(* IEC 61131-3 sources: cybercode_codesys_lib/src/signal/Analog, 5 files *)

(* ---- E_AlarmSetpoints.st ---- *)
TYPE E_AlarmSetpoints :
(
	Normal 	:= 0,
	L		:= 1,
	H		:= 2,
	LL		:= 3,
	HH		:= 4
);
END_TYPE

(* ---- FB_AnalogSignal4_20mA.st ---- *)
FUNCTION_BLOCK FB_AnalogSignal4_20mA EXTENDS FB_BasicAnalogSignal
VAR_INPUT
    rScaleMin : REAL := 0.0;        // Минимальное значение масштабируемого диапазона
    rScaleMax : REAL := 100.0;      // Максимальное значение масштабируемого диапазона
    xEnableRangeProtection : BOOL := TRUE;  // Включение защиты от выхода за диапазон
END_VAR
VAR_OUTPUT
END_VAR
VAR
    // Константы для токовой петли 4..20 мА
    _rCurrentMin : REAL := 4.0;     // Минимальный ток (мА)
    _rCurrentMax : REAL := 20.0;    // Максимальный ток (мА)

    // Состояние сигнала
    _xUnderrange : BOOL := FALSE;   // Сигнал ниже 4 мА
    _xOverrange : BOOL := FALSE;    // Сигнал выше 20 мА
    _xWireBreak : BOOL := FALSE;    // Обрыв линии (ток < 3.5 мА)
    _xOverload : BOOL := FALSE;     // Перегрузка (ток > 21 мА)

    // Пороговые значения для диагностики
    _rWireBreakThreshold : REAL := 3.5;    // Порог обрыва линии
    _rOverloadThreshold : REAL := 21.0;    // Порог перегрузки
END_VAR

// =====================================
// INPUT PROCESSING
// =====================================
ProcessRawValue();

// =====================================
// MAIN LOGIC
// =====================================
DiagnoseCurrent();

(* Обработка исходного токового сигнала *)
METHOD ProcessRawValue
VAR_INPUT
END_VAR
VAR
    rNormalizedCurrent : REAL;
END_VAR
    // Нормализация тока в диапазон 0..1
    IF (_rCurrentMax - _rCurrentMin) <> 0 THEN
        rNormalizedCurrent := (GetRawValue() - _rCurrentMin) / (_rCurrentMax - _rCurrentMin);
    ELSE
        rNormalizedCurrent := 0.0;
    END_IF

    // Масштабирование к заданному диапазону
    IF xEnableRangeProtection THEN
        // С ограничением диапазона
        rNormalizedCurrent := ClampToRange01(rNormalizedCurrent);
    END_IF

    SetProcessedValue(rScaleMin + rNormalizedCurrent * (rScaleMax - rScaleMin));
END_METHOD

(* Диагностика токового сигнала *)
METHOD PRIVATE DiagnoseCurrent
VAR_INPUT
END_VAR
VAR
    rCurrentValue : REAL;
END_VAR
    rCurrentValue := GetRawValue();

    // Проверка на обрыв линии
    _xWireBreak := rCurrentValue < _rWireBreakThreshold;

    // Проверка на перегрузку
    _xOverload := rCurrentValue > _rOverloadThreshold;

    // Проверка на выход за рабочий диапазон 4..20 мА
    _xUnderrange := (rCurrentValue < _rCurrentMin) AND NOT _xWireBreak;
    _xOverrange := (rCurrentValue > _rCurrentMax) AND NOT _xOverload;
END_METHOD

(* Получение масштабированного значения с учетом ошибок *)
METHOD GetScaledValue : REAL
VAR_INPUT
END_VAR
    IF _xWireBreak OR _xOverload THEN
        // При критических ошибках возвращаем минимальное значение
        GetScaledValue := rScaleMin;
    ELSE
        GetScaledValue := GetProcessedValue();
    END_IF
END_METHOD

(* Получение процентного значения (0..100%) *)
METHOD GetPercentValue : REAL
VAR_INPUT
END_VAR
VAR
    rNormalized : REAL;
END_VAR
    IF (rScaleMax - rScaleMin) <> 0 THEN
        rNormalized := (GetProcessedValue() - rScaleMin) / (rScaleMax - rScaleMin);
        GetPercentValue := rNormalized * 100.0;
    ELSE
        GetPercentValue := 0.0;
    END_IF
END_METHOD

(* Проверка на обрыв линии *)
METHOD IsWireBreak : BOOL
VAR_INPUT
END_VAR
    IsWireBreak := _xWireBreak;
END_METHOD

(* Проверка на перегрузку *)
METHOD IsOverload : BOOL
VAR_INPUT
END_VAR
    IsOverload := _xOverload;
END_METHOD

(* Проверка на нижний предел диапазона *)
METHOD IsUnderrange : BOOL
VAR_INPUT
END_VAR
    IsUnderrange := _xUnderrange;
END_METHOD

(* Проверка на верхний предел диапазона *)
METHOD IsOverrange : BOOL
VAR_INPUT
END_VAR
    IsOverrange := _xOverrange;
END_METHOD

(* Проверка на любую ошибку *)
METHOD HasError : BOOL
VAR_INPUT
END_VAR
    HasError := _xWireBreak OR _xOverload OR _xUnderrange OR _xOverrange;
END_METHOD

(* Установка масштабируемого диапазона *)
METHOD SetScaleRange
VAR_INPUT
    rMin : REAL;
    rMax : REAL;
END_VAR
    IF rMin < rMax THEN
        rScaleMin := rMin;
        rScaleMax := rMax;
    END_IF
END_METHOD

(* Получение минимального масштабируемого значения *)
METHOD GetScaleMin : REAL
VAR_INPUT
END_VAR
    GetScaleMin := rScaleMin;
END_METHOD

(* Получение максимального масштабируемого значения *)
METHOD GetScaleMax : REAL
VAR_INPUT
END_VAR
    GetScaleMax := rScaleMax;
END_METHOD

(* Сброс всех ошибок и состояний *)
METHOD Reset
VAR_INPUT
END_VAR
    // Вызов родительского сброса
    SUPER^.Reset();

    // Сброс локальных флагов
    _xUnderrange := FALSE;
    _xOverrange := FALSE;
    _xWireBreak := FALSE;
    _xOverload := FALSE;
END_METHOD

(* ========================================
   ЗАЩИЩЕННЫЕ МЕТОДЫ
   ======================================== *)

(* Ограничение значения в диапазоне 0..1 *)
METHOD PROTECTED ClampToRange01 : REAL
VAR_INPUT
    rValue : REAL;
END_VAR
    IF rValue < 0.0 THEN
        ClampToRange01 := 0.0;
    ELSIF rValue > 1.0 THEN
        ClampToRange01 := 1.0;
    ELSE
        ClampToRange01 := rValue;
    END_IF
END_METHOD

END_FUNCTION_BLOCK

(* ---- FB_BasicAnalogSignal.st ---- *)
FUNCTION_BLOCK ABSTRACT FB_BasicAnalogSignal
VAR_INPUT
    irRawValue : REAL;          // Исходное значение аналогового сигнала
END_VAR
VAR_OUTPUT
END_VAR
VAR
    _rProcessedValue : REAL;    // Обработанное значение сигнала
    _rMinValue : REAL := 0.0;   // Минимальное допустимое значение
    _rMaxValue : REAL := 100.0; // Максимальное допустимое значение
    _xOutOfRange : BOOL := FALSE; // Флаг выхода за пределы диапазона
END_VAR

// =====================================
// INPUT PROCESSING
// =====================================
ProcessRawValue();

// =====================================
// MAIN LOGIC
// =====================================
ValidateRange();

(* Получение исходного значения *)
METHOD GetRawValue : REAL
VAR_INPUT
END_VAR
    GetRawValue := irRawValue;
END_METHOD

(* Получение обработанного значения *)
METHOD GetProcessedValue : REAL
VAR_INPUT
END_VAR
    GetProcessedValue := _rProcessedValue;
END_METHOD

(* Получение статуса выхода за пределы диапазона *)
METHOD IsOutOfRange : BOOL
VAR_INPUT
END_VAR
    IsOutOfRange := _xOutOfRange;
END_METHOD

(* Получение минимального значения диапазона *)
METHOD GetMinValue : REAL
VAR_INPUT
END_VAR
    GetMinValue := _rMinValue;
END_METHOD

(* Получение максимального значения диапазона *)
METHOD GetMaxValue : REAL
VAR_INPUT
END_VAR
    GetMaxValue := _rMaxValue;
END_METHOD

(* Установка диапазона допустимых значений *)
METHOD SetRange
VAR_INPUT
    rMinValue : REAL;
    rMaxValue : REAL;
END_VAR
    IF rMinValue < rMaxValue THEN
        _rMinValue := rMinValue;
        _rMaxValue := rMaxValue;
    END_IF
END_METHOD

(* Проверка принадлежности значения к диапазону *)
METHOD IsInRange : BOOL
VAR_INPUT
    rValue : REAL;
END_VAR
    IsInRange := (rValue >= _rMinValue) AND (rValue <= _rMaxValue);
END_METHOD

(* Ограничение значения в пределах диапазона *)
METHOD ClampToRange : REAL
VAR_INPUT
    rValue : REAL;
END_VAR
    IF rValue < _rMinValue THEN
        ClampToRange := _rMinValue;
    ELSIF rValue > _rMaxValue THEN
        ClampToRange := _rMaxValue;
    ELSE
        ClampToRange := rValue;
    END_IF
END_METHOD

(* Сброс состояния функционального блока *)
METHOD Reset
VAR_INPUT
END_VAR
    _rProcessedValue := 0.0;
    _xOutOfRange := FALSE;
END_METHOD

(* ========================================
   АБСТРАКТНЫЕ МЕТОДЫ (должны быть переопределены в наследниках)
   ======================================== *)

(* Обработка исходного значения (абстрактный метод) *)
METHOD ABSTRACT ProcessRawValue
VAR_INPUT
END_VAR
END_METHOD

(* ========================================
   ЗАЩИЩЕННЫЕ МЕТОДЫ (для использования в наследниках)
   ======================================== *)

(* Проверка диапазона значений *)
METHOD PROTECTED ValidateRange
VAR_INPUT
END_VAR
    _xOutOfRange := NOT IsInRange(_rProcessedValue);
END_METHOD

(* Установка обработанного значения *)
METHOD PROTECTED SetProcessedValue
VAR_INPUT
    rValue : REAL;
END_VAR
    _rProcessedValue := rValue;
END_METHOD

END_FUNCTION_BLOCK

(* ---- FB_RangeDiagnostic_LH.st ---- *)
FUNCTION_BLOCK FB_RangeDiagnostic_LH
VAR_INPUT
    irValue : REAL;                     // Входное значение для контроля
    irSetpointL : REAL;         		// Уставка предупреждения низкого уровня
    irSetpointLL : REAL;        		// Уставка аварии низкого уровня
    irSetpointH : REAL;         		// Уставка предупреждения высокого уровня
    irSetpointHH : REAL;        		// Уставка аварии высокого уровня
    ixEnable : BOOL := TRUE;            // Разрешение работы блока
    irHysteresis : REAL := 1.0;         // Гистерезис для предотвращения дребезга
END_VAR
VAR_OUTPUT
    quAlarmCode : E_AlarmSetpoints;     // Код текущего состояния аварии/предупреждения
    qxAlarmActive : BOOL;               // TRUE = активна любая авария или предупреждение
    qxWarningActive : BOOL;             // TRUE = активно предупреждение (L или H)
    qxCriticalActive : BOOL;            // TRUE = активна критическая авария (LL или HH)
END_VAR
VAR
    _uPreviousAlarmCode : E_AlarmSetpoints := E_AlarmSetpoints.Normal;  // Предыдущий код аварии
    _xValidSetpoints : BOOL := TRUE;                                    // Флаг корректности уставок
    _rHysteresisValue : REAL;                                          // Текущее значение гистерезиса
END_VAR

// =====================================
// ВАЛИДАЦИЯ УСТАВОК
// =====================================
ValidateSetpoints();

// =====================================
// ОСНОВНАЯ ЛОГИКА ОПРЕДЕЛЕНИЯ АВАРИЙ
// =====================================
IF ixEnable AND _xValidSetpoints THEN
    ProcessAlarms();
ELSE
    // При отключении или некорректных уставках - сброс в нормальное состояние
    quAlarmCode := E_AlarmSetpoints.Normal;
END_IF

// =====================================
// ОБНОВЛЕНИЕ ВЫХОДНЫХ СИГНАЛОВ
// =====================================
UpdateOutputs();

(* Валидация корректности уставок *)
METHOD PRIVATE ValidateSetpoints
VAR_INPUT
END_VAR
    // Проверяем логическую корректность уставок: LL < L < H < HH
    _xValidSetpoints := (irSetpointLL <= irSetpointL) AND
                       (irSetpointL < irSetpointH) AND
                       (irSetpointH <= irSetpointHH);

    // Гистерезис не может быть отрицательным
    IF irHysteresis < 0 THEN
        _rHysteresisValue := 0;
    ELSE
        _rHysteresisValue := irHysteresis;
    END_IF
END_METHOD

(* Основная логика обработки аварий с гистерезисом *)
METHOD PRIVATE ProcessAlarms
VAR_INPUT
END_VAR
    // Сохраняем предыдущее состояние
    _uPreviousAlarmCode := quAlarmCode;

    // Определяем новое состояние на основе текущего значения
    IF irValue <= irSetpointLL THEN
        quAlarmCode := E_AlarmSetpoints.LL;
    ELSIF irValue <= irSetpointL THEN
        quAlarmCode := E_AlarmSetpoints.L;
    ELSIF irValue >= irSetpointHH THEN
        quAlarmCode := E_AlarmSetpoints.HH;
    ELSIF irValue >= irSetpointH THEN
        quAlarmCode := E_AlarmSetpoints.H;
    ELSE
        // Проверяем гистерезис для возврата в нормальное состояние
        ApplyHysteresis();
    END_IF
END_METHOD

(* Применение гистерезиса для предотвращения дребезга *)
METHOD PRIVATE ApplyHysteresis
VAR_INPUT
END_VAR
    // Применяем гистерезис только при возврате к нормальному состоянию
    CASE _uPreviousAlarmCode OF
        E_AlarmSetpoints.LL:
            // Возврат из LL возможен только при превышении LL + гистерезис
            IF irValue > (irSetpointLL + _rHysteresisValue) THEN
                quAlarmCode := E_AlarmSetpoints.Normal;
            ELSE
                quAlarmCode := E_AlarmSetpoints.LL;
            END_IF

        E_AlarmSetpoints.L:
            // Возврат из L возможен только при превышении L + гистерезис
            IF irValue > (irSetpointL + _rHysteresisValue) THEN
                quAlarmCode := E_AlarmSetpoints.Normal;
            ELSE
                quAlarmCode := E_AlarmSetpoints.L;
            END_IF

        E_AlarmSetpoints.H:
            // Возврат из H возможен только при снижении ниже H - гистерезис
            IF irValue < (irSetpointH - _rHysteresisValue) THEN
                quAlarmCode := E_AlarmSetpoints.Normal;
            ELSE
                quAlarmCode := E_AlarmSetpoints.H;
            END_IF

        E_AlarmSetpoints.HH:
            // Возврат из HH возможен только при снижении ниже HH - гистерезис
            IF irValue < (irSetpointHH - _rHysteresisValue) THEN
                quAlarmCode := E_AlarmSetpoints.Normal;
            ELSE
                quAlarmCode := E_AlarmSetpoints.HH;
            END_IF

        E_AlarmSetpoints.Normal:
            // Остаемся в нормальном состоянии
            quAlarmCode := E_AlarmSetpoints.Normal;
    END_CASE
END_METHOD

(* Обновление выходных сигналов *)
METHOD PRIVATE UpdateOutputs
VAR_INPUT
END_VAR
    // Флаг активности любой аварии или предупреждения
    qxAlarmActive := (quAlarmCode <> E_AlarmSetpoints.Normal);

    // Флаг активности предупреждений (L, H)
    qxWarningActive := (quAlarmCode = E_AlarmSetpoints.L) OR
                      (quAlarmCode = E_AlarmSetpoints.H);

    // Флаг активности критических аварий (LL, HH)
    qxCriticalActive := (quAlarmCode = E_AlarmSetpoints.LL) OR
                       (quAlarmCode = E_AlarmSetpoints.HH);
END_METHOD

(* ========================================
   МЕТОДЫ ПОЛУЧЕНИЯ ИНФОРМАЦИИ
   ======================================== *)

(* Получение текущего кода аварии *)
METHOD GetAlarmCode : E_AlarmSetpoints
VAR_INPUT
END_VAR
    GetAlarmCode := quAlarmCode;
END_METHOD

(* Получение входного значения *)
METHOD GetCurrentValue : REAL
VAR_INPUT
END_VAR
    GetCurrentValue := irValue;
END_METHOD

(* Проверка состояния "в норме" *)
METHOD IsNormal : BOOL
VAR_INPUT
END_VAR
    IsNormal := (quAlarmCode = E_AlarmSetpoints.Normal);
END_METHOD

(* Проверка активности низких аварий (L или LL) *)
METHOD IsLowAlarm : BOOL
VAR_INPUT
END_VAR
    IsLowAlarm := (quAlarmCode = E_AlarmSetpoints.L) OR
                  (quAlarmCode = E_AlarmSetpoints.LL);
END_METHOD

(* Проверка активности высоких аварий (H или HH) *)
METHOD IsHighAlarm : BOOL
VAR_INPUT
END_VAR
    IsHighAlarm := (quAlarmCode = E_AlarmSetpoints.H) OR
                   (quAlarmCode = E_AlarmSetpoints.HH);
END_METHOD

(* Проверка корректности уставок *)
METHOD AreSetpointsValid : BOOL
VAR_INPUT
END_VAR
    AreSetpointsValid := _xValidSetpoints;
END_METHOD

(* Получение расстояния до ближайшей уставки *)
METHOD GetDistanceToNearestSetpoint : REAL
VAR_INPUT
END_VAR
VAR
    rDistanceToL : REAL;
    rDistanceToLL : REAL;
    rDistanceToH : REAL;
    rDistanceToHH : REAL;
    rMinDistance : REAL;
END_VAR
    rDistanceToL := ABS(irValue - irSetpointL);
    rDistanceToLL := ABS(irValue - irSetpointLL);
    rDistanceToH := ABS(irValue - irSetpointH);
    rDistanceToHH := ABS(irValue - irSetpointHH);

    rMinDistance := rDistanceToL;
    IF rDistanceToLL < rMinDistance THEN rMinDistance := rDistanceToLL; END_IF
    IF rDistanceToH < rMinDistance THEN rMinDistance := rDistanceToH; END_IF
    IF rDistanceToHH < rMinDistance THEN rMinDistance := rDistanceToHH; END_IF

    GetDistanceToNearestSetpoint := rMinDistance;
END_METHOD

(* ========================================
   МЕТОДЫ НАСТРОЙКИ
   ======================================== *)

(* Установка всех уставок одновременно *)
METHOD SetAllSetpoints
VAR_INPUT
    rLL : REAL;     // Авария низкого уровня
    rL : REAL;      // Предупреждение низкого уровня
    rH : REAL;      // Предупреждение высокого уровня
    rHH : REAL;     // Авария высокого уровня
END_VAR
    // Проверяем корректность перед установкой
    IF (rLL <= rL) AND (rL < rH) AND (rH <= rHH) THEN
        irSetpointLL := rLL;
        irSetpointL := rL;
        irSetpointH := rH;
        irSetpointHH := rHH;
    END_IF
END_METHOD

(* Установка симметричных уставок относительно центрального значения *)
METHOD SetSymmetricSetpoints
VAR_INPUT
    rCenterValue : REAL;    // Центральное (номинальное) значение
    rWarningOffset : REAL;  // Смещение для предупреждений (L, H)
    rAlarmOffset : REAL;    // Смещение для аварий (LL, HH)
END_VAR
    IF (rWarningOffset >= 0) AND (rAlarmOffset >= rWarningOffset) THEN
        irSetpointL := rCenterValue - rWarningOffset;
        irSetpointLL := rCenterValue - rAlarmOffset;
        irSetpointH := rCenterValue + rWarningOffset;
        irSetpointHH := rCenterValue + rAlarmOffset;
    END_IF
END_METHOD

(* Установка уставок в процентах от диапазона *)
METHOD SetSetpointsPercent
VAR_INPUT
    rMinValue : REAL;       // Минимальное значение диапазона
    rMaxValue : REAL;       // Максимальное значение диапазона
    rLLPercent : REAL;      // Процент для LL (0..100)
    rLPercent : REAL;       // Процент для L (0..100)
    rHPercent : REAL;       // Процент для H (0..100)
    rHHPercent : REAL;      // Процент для HH (0..100)
END_VAR
VAR
    rRange : REAL;
END_VAR
    IF (rMinValue < rMaxValue) AND
       (rLLPercent <= rLPercent) AND (rLPercent < rHPercent) AND (rHPercent <= rHHPercent) AND
       (rLLPercent >= 0) AND (rHHPercent <= 100) THEN

        rRange := rMaxValue - rMinValue;
        irSetpointLL := rMinValue + (rRange * rLLPercent / 100.0);
        irSetpointL := rMinValue + (rRange * rLPercent / 100.0);
        irSetpointH := rMinValue + (rRange * rHPercent / 100.0);
        irSetpointHH := rMinValue + (rRange * rHHPercent / 100.0);
    END_IF
END_METHOD

(* ========================================
   СЕРВИСНЫЕ МЕТОДЫ
   ======================================== *)

(* Полный сброс состояния *)
METHOD Reset
VAR_INPUT
END_VAR
    quAlarmCode := E_AlarmSetpoints.Normal;
    _uPreviousAlarmCode := E_AlarmSetpoints.Normal;
    qxAlarmActive := FALSE;
    qxWarningActive := FALSE;
    qxCriticalActive := FALSE;
END_METHOD

(* Принудительная установка состояния "норма" *)
METHOD ForceNormal
VAR_INPUT
END_VAR
    quAlarmCode := E_AlarmSetpoints.Normal;
    _uPreviousAlarmCode := E_AlarmSetpoints.Normal;
    UpdateOutputs();
END_METHOD

END_FUNCTION_BLOCK

(* ---- FB_UniversalAnalogSignal .st ---- *)
FUNCTION_BLOCK FB_UniversalAnalogSignal EXTENDS FB_BasicAnalogSignal
VAR_INPUT
    // Диапазон входного аналогового сигнала
    rInputMin : REAL := 0.0;        // Минимальное значение входного сигнала
    rInputMax : REAL := 10.0;       // Максимальное значение входного сигнала

    // Диапазон масштабирования (выходные инженерные единицы)
    rScaleMin : REAL := 0.0;        // Минимальное значение масштабированного диапазона
    rScaleMax : REAL := 100.0;      // Максимальное значение масштабированного диапазона

    // Настройки
    xEnableRangeProtection : BOOL := TRUE;  // Включение защиты от выхода за диапазон
    xEnableDiagnostics : BOOL := TRUE;      // Включение диагностики сигнала
END_VAR
VAR_OUTPUT
END_VAR
VAR
    // Диагностика сигнала
    _xSignalUnderrange : BOOL := FALSE;     // Сигнал ниже минимума входного диапазона
    _xSignalOverrange : BOOL := FALSE;      // Сигнал выше максимума входного диапазона

    // Пороги для расширенной диагностики (в % от диапазона)
    _rUnderrangeThreshold : REAL := 5.0;    // Порог для определения критически низкого сигнала
    _rOverrangeThreshold : REAL := 5.0;     // Порог для определения критически высокого сигнала

    // Расширенная диагностика
    _xCriticalLow : BOOL := FALSE;          // Критически низкий сигнал
    _xCriticalHigh : BOOL := FALSE;         // Критически высокий сигнал

    // Вычисленные значения
    _rNormalizedValue : REAL := 0.0;        // Нормализованное значение (0..1)
    _rPercentValue : REAL := 0.0;           // Процентное значение (0..100%)
END_VAR

// =====================================
// ОБРАБОТКА ВХОДНОГО СИГНАЛА
// =====================================
ProcessRawValue();

// =====================================
// ДИАГНОСТИКА
// =====================================
IF xEnableDiagnostics THEN
    DiagnoseSignal();
END_IF

// =====================================
// ВЫЧИСЛЕНИЕ ДОПОЛНИТЕЛЬНЫХ ЗНАЧЕНИЙ
// =====================================
CalculateAdditionalValues();

(* Обработка исходного сигнала и масштабирование *)
METHOD ProcessRawValue
VAR_INPUT
END_VAR
VAR
    rInputRange : REAL;
    rScaleRange : REAL;
    rRawSignal : REAL;
END_VAR
    rRawSignal := GetRawValue();

    // Вычисление диапазонов
    rInputRange := rInputMax - rInputMin;
    rScaleRange := rScaleMax - rScaleMin;

    // Проверка корректности диапазонов
    IF (rInputRange = 0) OR (rScaleRange = 0) THEN
        SetProcessedValue(rScaleMin);
        RETURN;
    END_IF

    // Нормализация входного сигнала (приведение к диапазону 0..1)
    _rNormalizedValue := (rRawSignal - rInputMin) / rInputRange;

    // Применение ограничений если включена защита
    IF xEnableRangeProtection THEN
        _rNormalizedValue := LimitTo01(_rNormalizedValue);
    END_IF

    // Масштабирование к выходному диапазону
    SetProcessedValue(rScaleMin + _rNormalizedValue * rScaleRange);
END_METHOD

(* Диагностика входного сигнала *)
METHOD PRIVATE DiagnoseSignal
VAR_INPUT
END_VAR
VAR
    rRawSignal : REAL;
    rInputRange : REAL;
    rCriticalLowLimit : REAL;
    rCriticalHighLimit : REAL;
END_VAR
    rRawSignal := GetRawValue();
    rInputRange := rInputMax - rInputMin;

    // Базовая диагностика диапазона
    _xSignalUnderrange := rRawSignal < rInputMin;
    _xSignalOverrange := rRawSignal > rInputMax;

    // Расширенная диагностика (критические пределы)
    IF rInputRange <> 0 THEN
        // Вычисление критических порогов
        rCriticalLowLimit := rInputMin - (rInputRange * _rUnderrangeThreshold / 100.0);
        rCriticalHighLimit := rInputMax + (rInputRange * _rOverrangeThreshold / 100.0);

        _xCriticalLow := rRawSignal < rCriticalLowLimit;
        _xCriticalHigh := rRawSignal > rCriticalHighLimit;
    END_IF
END_METHOD

(* Вычисление дополнительных значений *)
METHOD PRIVATE CalculateAdditionalValues
VAR_INPUT
END_VAR
    // Процентное значение относительно масштабированного диапазона
    IF (rScaleMax - rScaleMin) <> 0 THEN
        _rPercentValue := ((GetProcessedValue() - rScaleMin) / (rScaleMax - rScaleMin)) * 100.0;
    ELSE
        _rPercentValue := 0.0;
    END_IF
END_METHOD

(* ========================================
   МЕТОДЫ ПОЛУЧЕНИЯ ЗНАЧЕНИЙ
   ======================================== *)

(* Получение масштабированного значения *)
METHOD GetScaledValue : REAL
VAR_INPUT
END_VAR
    // При критических ошибках возвращаем безопасное значение
    IF _xCriticalLow OR _xCriticalHigh THEN
        GetScaledValue := rScaleMin;
    ELSE
        GetScaledValue := GetProcessedValue();
    END_IF
END_METHOD

(* Получение нормализованного значения (0..1) *)
METHOD GetNormalizedValue : REAL
VAR_INPUT
END_VAR
    GetNormalizedValue := _rNormalizedValue;
END_METHOD

(* Получение процентного значения *)
METHOD GetPercentValue : REAL
VAR_INPUT
END_VAR
    GetPercentValue := _rPercentValue;
END_METHOD

(* Получение процента относительно входного диапазона *)
METHOD GetInputRangePercent : REAL
VAR_INPUT
END_VAR
    IF (rInputMax - rInputMin) <> 0 THEN
        GetInputRangePercent := ((GetRawValue() - rInputMin) / (rInputMax - rInputMin)) * 100.0;
    ELSE
        GetInputRangePercent := 0.0;
    END_IF
END_METHOD

(* ========================================
   МЕТОДЫ ДИАГНОСТИКИ
   ======================================== *)

(* Проверка выхода за нижний предел *)
METHOD IsUnderrange : BOOL
VAR_INPUT
END_VAR
    IsUnderrange := _xSignalUnderrange;
END_METHOD

(* Проверка выхода за верхний предел *)
METHOD IsOverrange : BOOL
VAR_INPUT
END_VAR
    IsOverrange := _xSignalOverrange;
END_METHOD

(* Проверка критически низкого сигнала *)
METHOD IsCriticalLow : BOOL
VAR_INPUT
END_VAR
    IsCriticalLow := _xCriticalLow;
END_METHOD

(* Проверка критически высокого сигнала *)
METHOD IsCriticalHigh : BOOL
VAR_INPUT
END_VAR
    IsCriticalHigh := _xCriticalHigh;
END_METHOD

(* Проверка на любую ошибку *)
METHOD HasError : BOOL
VAR_INPUT
END_VAR
    HasError := _xSignalUnderrange OR _xSignalOverrange OR _xCriticalLow OR _xCriticalHigh;
END_METHOD

(* Проверка на критическую ошибку *)
METHOD HasCriticalError : BOOL
VAR_INPUT
END_VAR
    HasCriticalError := _xCriticalLow OR _xCriticalHigh;
END_METHOD

(* Проверка нахождения в допустимом диапазоне *)
METHOD IsInValidRange : BOOL
VAR_INPUT
END_VAR
    IsInValidRange := NOT (_xSignalUnderrange OR _xSignalOverrange);
END_METHOD

(* ========================================
   МЕТОДЫ НАСТРОЙКИ
   ======================================== *)

(* Установка входного диапазона *)
METHOD SetInputRange
VAR_INPUT
    rMin : REAL;
    rMax : REAL;
END_VAR
    IF rMin < rMax THEN
        rInputMin := rMin;
        rInputMax := rMax;
    END_IF
END_METHOD

(* Установка диапазона масштабирования *)
METHOD SetScaleRange
VAR_INPUT
    rMin : REAL;
    rMax : REAL;
END_VAR
    IF rMin < rMax THEN
        rScaleMin := rMin;
        rScaleMax := rMax;
    END_IF
END_METHOD

(* Установка порогов критической диагностики *)
METHOD SetDiagnosticThresholds
VAR_INPUT
    rUnderrangePercent : REAL;  // Процент от диапазона для критически низкого
    rOverrangePercent : REAL;   // Процент от диапазона для критически высокого
END_VAR
    IF (rUnderrangePercent >= 0) AND (rUnderrangePercent <= 100) THEN
        _rUnderrangeThreshold := rUnderrangePercent;
    END_IF

    IF (rOverrangePercent >= 0) AND (rOverrangePercent <= 100) THEN
        _rOverrangeThreshold := rOverrangePercent;
    END_IF
END_METHOD

(* Конфигурация для стандартных типов сигналов *)
METHOD ConfigureAs4_20mA
VAR_INPUT
    rProcessMin : REAL := 0.0;   // Минимальное значение процесса
    rProcessMax : REAL := 100.0; // Максимальное значение процесса
END_VAR
    SetInputRange(4.0, 20.0);
    SetScaleRange(rProcessMin, rProcessMax);
    SetDiagnosticThresholds(12.5, 5.0);  // 3.5мА и 21мА соответственно
END_METHOD

METHOD ConfigureAs0_10V
VAR_INPUT
    rProcessMin : REAL := 0.0;
    rProcessMax : REAL := 100.0;
END_VAR
    SetInputRange(0.0, 10.0);
    SetScaleRange(rProcessMin, rProcessMax);
    SetDiagnosticThresholds(5.0, 5.0);
END_METHOD

METHOD ConfigureAs0_20mA
VAR_INPUT
    rProcessMin : REAL := 0.0;
    rProcessMax : REAL := 100.0;
END_VAR
    SetInputRange(0.0, 20.0);
    SetScaleRange(rProcessMin, rProcessMax);
    SetDiagnosticThresholds(5.0, 5.0);
END_METHOD

METHOD ConfigureAsPt100
VAR_INPUT
    rTempMin : REAL := -50.0;   // Минимальная температура
    rTempMax : REAL := 200.0;   // Максимальная температура
END_VAR
    // Примерные значения сопротивления для Pt100
    SetInputRange(80.31, 175.86);  // Сопротивление при -50°C и 200°C
    SetScaleRange(rTempMin, rTempMax);
    SetDiagnosticThresholds(2.0, 2.0);
END_METHOD

(* ========================================
   МЕТОДЫ ПОЛУЧЕНИЯ ИНФОРМАЦИИ О КОНФИГУРАЦИИ
   ======================================== *)

(* Получение минимума входного диапазона *)
METHOD GetInputMin : REAL
VAR_INPUT
END_VAR
    GetInputMin := rInputMin;
END_METHOD

(* Получение максимума входного диапазона *)
METHOD GetInputMax : REAL
VAR_INPUT
END_VAR
    GetInputMax := rInputMax;
END_METHOD

(* Получение минимума масштабированного диапазона *)
METHOD GetScaleMin : REAL
VAR_INPUT
END_VAR
    GetScaleMin := rScaleMin;
END_METHOD

(* Получение максимума масштабированного диапазона *)
METHOD GetScaleMax : REAL
VAR_INPUT
END_VAR
    GetScaleMax := rScaleMax;
END_METHOD

(* Получение размаха входного диапазона *)
METHOD GetInputSpan : REAL
VAR_INPUT
END_VAR
    GetInputSpan := rInputMax - rInputMin;
END_METHOD

(* Получение размаха масштабированного диапазона *)
METHOD GetScaleSpan : REAL
VAR_INPUT
END_VAR
    GetScaleSpan := rScaleMax - rScaleMin;
END_METHOD

(* ========================================
   ВСПОМОГАТЕЛЬНЫЕ МЕТОДЫ
   ======================================== *)

(* Полный сброс состояния *)
METHOD Reset
VAR_INPUT
END_VAR
    // Вызов родительского метода
    SUPER^.Reset();

    // Сброс локальных флагов диагностики
    _xSignalUnderrange := FALSE;
    _xSignalOverrange := FALSE;
    _xCriticalLow := FALSE;
    _xCriticalHigh := FALSE;

    // Сброс вычисленных значений
    _rNormalizedValue := 0.0;
    _rPercentValue := 0.0;
END_METHOD

(* Ограничение значения в диапазоне 0..1 *)
METHOD PRIVATE LimitTo01 : REAL
VAR_INPUT
    rValue : REAL;
END_VAR
    IF rValue < 0.0 THEN
        LimitTo01 := 0.0;
    ELSIF rValue > 1.0 THEN
        LimitTo01 := 1.0;
    ELSE
        LimitTo01 := rValue;
    END_IF
END_METHOD

END_FUNCTION_BLOCK
